{attribute addProperty BoxType "EK1100-0000-0018"}
{attribute addProperty Id "Beckhoff_ELM3xxx_0030EK1122Beckhoff_ELM3xxx_0030EK1122_7F195F23162A_0001_ELM3002_0030_0017ELM3002_1C598C2535244A_0002_ELM3002_0030_0018ELM3002_1C598C2535244A_0003_ELM3004_0030_0018ELM3004_EF18820948060A_0004_ELM3004_0030_0019ELM3004_EF18820948060A_0005_ELM3502_0030_0019ELM3502_1C598C2535244A_0006_ELM3504_0030_0019ELM3504_EF18820948060"}
{attribute addProperty CRC "127424737"}
{attribute addProperty SizeInBites "2512"}
{attribute addProperty SizeInBytes "314"}
TYPE Beckhoff_ELM3xxx_0030_079858E1 EXTENDS EK1100_179A0949 :
STRUCT
	{attribute addProperty Name "Beckhoff_ELM3xxx_0030EK1122"}
	Beckhoff_ELM3xxx_0030EK1122 : Beckhoff_ELM3xxx_0030EK1122_7F195F23;
	{attribute addProperty Name "A_0001_ELM3002_0030_0017"}
	A_0001_ELM3002_0030_0017 : ELM3002_1C598C25;
	{attribute addProperty Name "A_0002_ELM3002_0030_0018"}
	A_0002_ELM3002_0030_0018 : ELM3002_1C598C25;
	{attribute addProperty Name "A_0003_ELM3004_0030_0018"}
	A_0003_ELM3004_0030_0018 : ELM3004_EF188209;
	{attribute addProperty Name "A_0004_ELM3004_0030_0019"}
	A_0004_ELM3004_0030_0019 : ELM3004_EF188209;
	{attribute addProperty Name "A_0005_ELM3502_0030_0019"}
	A_0005_ELM3502_0030_0019 : ELM3502_1C598C25;
	{attribute addProperty Name "A_0006_ELM3504_0030_0019"}
	A_0006_ELM3504_0030_0019 : ELM3504_EF188209;
END_STRUCT
END_TYPE

(* stored: Version 1.2.0.0, ProductVersion 3.1.4024.9
   DUT Beckhoff_ELM3xxx_0030_079858E1: Id {4f86f6ec-b031-4670-be9a-2631eaaea4f6} *)
